{attribute 'qualified_only'}
{attribute 'strict'}
TYPE E_Transfer :
(
	IDLE := 0,
	LOAD,
	UNLOAD
);
END_TYPE

(* stored: Version 1.1.0.1, ProductVersion 3.1.4024.12
   DUT E_Transfer: Id {17e10a8e-f8f0-4839-9d15-166482917a84} *)
